// FB_SafePower sets contactor and lamp for one safety power output
FUNCTION_BLOCK FB_SafePower
VAR_INPUT
	bSwitchPower 		: BOOL; // switch is set to ON
	bHasPower			: BOOL; // contactor has power (Safety OK)
END_VAR
VAR_OUTPUT
	bLightSelectPower 	: BOOL; // lamp
	bSetSafetyPower		: BOOL; // bSwitchPower
END_VAR

VAR
//	fbBlink: FB_Blink;
END_VAR

bSetSafetyPower := bSwitchPower;

IF bSetSafetyPower AND bHasPower THEN
	bLightSelectPower := TRUE;
//ELSIF bSetSafetyPower AND NOT bHasPower THEN
//	fbBlink(bEnable:= TRUE, bOut=> bLightSelectPower);
ELSE
	bLightSelectPower := FALSE;
END_IF

END_FUNCTION_BLOCK

(* stored: Version 1.1.0.1, ProductVersion 3.1.4024.10
   POU FB_SafePower: Id {9e63c281-7858-4abc-b5cd-14504f4701fe}, SpecialFunc None *)
